Staubli VAL3: ros_server.pjx

--- ros_server.pjx ---
Parameters version=s7.7.2 stackSize=5000 millimeterUnit=true
Program file=dataReceiver.pgx
Program file=dataStreamer.pgx
Program file=decodeMsgBody.pgx
Program file=decodeMsgHeader.pgx
Program file=decTrajPt.pgx
Program file=decTrajPtFull.pgx
Program file=encodeAck.pgx
Program file=encodeJState.pgx
Program file=encodeStatus.pgx
Program file=encPrefixHeader.pgx
Program file=encTrajPtAck.pgx
Program file=encTrajPtFAck.pgx
Program file=fetchStatus.pgx
Program file=initParams.pgx
Program file=motionControl.pgx
Program file=pushMotion.pgx
Program file=recvData.pgx
Program file=recvHeartbeat.pgx
Program file=recvMsgBody.pgx
Program file=recvMsgHeader.pgx
Program file=recvTrajPt.pgx
Program file=recvTrajPtFull.pgx
Program file=screenUpdate.pgx
Program file=sendAck.pgx
Program file=sendData.pgx
Program file=sendRosMsg.pgx
Program file=setupRosMsgs.pgx
Program file=start.pgx
Program file=stop.pgx
Program file=toJointArrayRad.pgx
Program file=toJointRxDeg.pgx
Data file=ros_server.dtx
Library alias=libQueueFuncs path=Disk://ros_libs/QueueFuncs/QueueFuncs.pjx
Type name=RosSimpleMsg path=Disk://ros_libs/RosSimpleMsg/RosSimpleMsg.pjx
Type name=RobotStatusMsg path=Disk://ros_libs/RobotStatusMsg/RobotStatusMsg.pjx
Type name=JointStateMsg path=Disk://ros_libs/JointStateMsg/JointStateMsg.pjx
Type name=JointTrajPtMsg path=Disk://ros_libs/JointTrajPtMsg/JointTrajPtMsg.pjx
Type name=JointTrajPtFMsg path=Disk://ros_libs/JointTrajPtFMsg/JointTrajPtFMsg.pjx
Type name=JointFbkMsg path=Disk://ros_libs/JointFbkMsg/JointFbkMsg.pjx
Type name=MotionCmd path=Disk://ros_libs/MotionCmd/MotionCmd.pjx
Type name=Header path=Disk://ros_libs/Header/Header.pjx
Type name=Prefix path=Disk://ros_libs/Prefix/Prefix.pjx
Type name=Body path=Disk://ros_libs/Body/Body.pjx
Type name=Queue path=Disk://ros_libs/Queue/Queue.pjx

--- ros_server.dtx ---
public bool bFbkOverrun
public bool bMotionOverrun
public jointRx jCurrPose
public num nCounter
public num nFbkPeriod = 0.032
num nMotionPeriod = 0.012
public sio siTcpIpFbk = {link=Socket\Feedback}
public sio siTcpIpMotion = {link=Socket\Motion}
public string sStreamTaskName = "publisher"
public string sMotionTaskName
public bool bSendData
public RosSimpleMsg rosGenericMsg
  [0]
    Header header
      [0]
        num nMsgType
        num nCommType
        num nReplyCode
        num nData[12]
    Prefix prefix
      [0]
        num nLength
        num nData[4]
public jointRx jDesiredPose
public tool tTool = {fatherId=flange[0], ioLink=valve1}
public string sTrajPtTaskName
public bool bTrajPtOverrun
public RobotStatusMsg rosStatusMsg
  [0]
    Body body
      [0]
        num nData[28]
    Header header
      [0]
        num nMsgType
        num nCommType
        num nReplyCode
        num nData[12]
    Prefix prefix
      [0]
        num nLength
        num nData[4]
    RobotStatus robotStatus
      [0]
        num nDrivesPowered
        num nEStopped
        num nErrorCode
        num nInError
        num nInMotion
        num nMode
        num nMotionPossible
public JointStateMsg rosJointMsg
  [0]
    Header header
      [0]
        num nMsgType
        num nCommType
        num nReplyCode
        num nData[12]
    Body body
      [0]
        num nData[44]
    JointState jointState
      [0]
        num nSeq
        num nJoints[10]
    Prefix prefix
      [0]
        num nLength
        num nData[4]
public JointTrajPtMsg rosTrajPtMsg
  [0]
    Header header
      [0]
        num nMsgType
        num nCommType
        num nReplyCode
        num nData[12]
    JointTrajPt jointTrajPt
      [0]
        num nSeq
        num nJoints[10]
        num nVelocity
        num nDuration
    Prefix prefix
      [0]
        num nLength
        num nData[4]
    Body body
      [0]
        num nData[52]
public bool bRecvData
public JointTrajPtFMsg rosTrajPtFMsg
  [0]
    Header header
      [0]
        num nMsgType
        num nCommType
        num nReplyCode
        num nData[12]
    Prefix prefix
      [0]
        num nLength
        num nData[4]
    JointTrajPtFull jointTrajPtFull
      [0]
        num nRobotId
        num nSeq
        num nValidFields
        num nTime
        num nPositions[10]
        num nVelocities[10]
        num nAccelerations[10]
    Body body
      [0]
        num nData[136]
public JointFbkMsg rosJointFbkMsg
  [0]
    Header header
      [0]
        num nMsgType
        num nCommType
        num nReplyCode
        num nData[12]
    Prefix prefix
      [0]
        num nLength
        num nData[4]
    JointFeedback jointFeedback
      [0]
        num nRobotId
        num nValidFields
        num nTime
        num nPositions[10]
        num nVelocities[10]
        num nAccelerations[10]
    Body body
      [0]
        num nData[132]
public JointTrajPtFMsg rosTrajPtFAck
  [0]
    Header header
      [0]
        num nMsgType
        num nCommType
        num nReplyCode
        num nData[12]
    Prefix prefix
      [0]
        num nLength
        num nData[4]
    JointTrajPtFull jointTrajPtFull
      [0]
        num nRobotId
        num nSeq
        num nValidFields
        num nTime
        num nPositions[10]
        num nVelocities[10]
        num nAccelerations[10]
    Body body
      [0]
        num nData[136]
public JointTrajPtMsg rosTrajPtAck
  [0]
    Header header
      [0]
        num nMsgType
        num nCommType
        num nReplyCode
        num nData[12]
    JointTrajPt jointTrajPt
      [0]
        num nSeq
        num nJoints[10]
        num nVelocity
        num nDuration
    Prefix prefix
      [0]
        num nLength
        num nData[4]
    Body body
      [0]
        num nData[52]
public bool bScreenOverrun
public string sScreenTaskName
public num nScreenUpdate
public num nTrajReception
public num nInConnFlag
public num nOutConnFlag
public num nDebugStatus
public screen scDebug
public screen scMonitor
public string sHtbtTaskName
public num nMsgRecvState
public num nPtsPopped
public bool bStopNow
public MotionBuffer mTrajPt
  [0]
    mdesc mDesc = {leave=0, reach=0}
    num nDuration
    num nSequence
    jointRx jJointRx
public num nMotionProgress
public num nMoveId
public num nMovePts
public num nElapsedTime
public num nHeaderTime
public num nOtherTime
public num nStartTime
public bool bOverwriteVel
public num nKey

--- start.pgx ---
program start()
  local num l_nFbkPeriod
  local num l_nMotionPeriod
  local num l_nTrajPeriod
  local num l_nScreenUpdate
begin
  // Copyright (c) 2016, Ocado Technology - Robotics Research Team
  //
  // Licensed under the Apache License, Version 2.0 (the "License");
  // you may not use this file except in compliance with the License.
  // You may obtain a copy of the License at
  //
  //     http://www.apache.org/licenses/LICENSE-2.0
  //
  // Unless required by applicable law or agreed to in writing, software
  // distributed under the License is distributed on an "AS IS" BASIS,
  // WITHOUT WARRANTIES OR CONDITIONS OF ANY KIND, either express or implied.
  // See the License for the specific language governing permissions and
  // limitations under the License.



  // feedback task will run every 20ms (50Hz)
  l_nFbkPeriod=0.02
  //l_nFbkPeriod = 0.032 // 30Hz
  //l_nFbkPeriod = 0.05  // 20Hz
  //l_nFbkPeriod = 1.0   //  1Hz

  // motion control task will run every 4ms (250Hz)
  l_nMotionPeriod = 0.004
  //l_nMotionPeriod=0.012  // 83Hz
  //l_nMotionPeriod = 0.05 // 20Hz

  // data (trajectory) reception task will run every 4ms (250Hz)
  l_nTrajPeriod = 0.004
  // not in use at the moment
  l_nScreenUpdate = 1.0

  sStreamTaskName = "streamerTask"
  sTrajPtTaskName = "trajPtTask"
  sMotionTaskName = "motionTask"
  sScreenTaskName = "screenTask"
  sHtbtTaskName = "htbtTask"

  // initialise TCP/IP parameters
  call initParams()
  // setup prefix and header of ROS messages
  call setupRosMsgs()

  // socket connection status flags: initially disconnected
  nInConnFlag = 0
  nOutConnFlag = 0

  // flag defining whether velocity to be overwritten to max. vel.
  bOverwriteVel = false

  nPtsPopped = 0
  nMovePts = 0

  // flush buffer of incoming socket
  clearBuffer(siTcpIpMotion)
  // flush buffer of outgoing socket
  clearBuffer(siTcpIpFbk)

  // check if robot is not in emergency stop and wait until estop is reset
  if (esStatus() == 2)
    popUpMsg("Please reset E-Stop")
    wait(esStatus() < 2)
  endIf

  // before anything else, enable power (only works if robot is in remote mode)
  if (!isPowered())
    if (workingMode() >= 4)
      do
        enablePower()
        delay(2)
      until isPowered()
    else
      popUpMsg("Power must be enabled manually")
    endIf
  endIf

  // reset motion, potentially setting a start joint position for calling autoConnect() in the future
  resetMotion()

  // create joint state and robot status streamer task to send data to industrial_robot_client
  taskCreateSync sStreamTaskName, l_nFbkPeriod, bFbkOverrun, dataStreamer()

  // create trajectory point task to receive data from industrial_robot_client
  taskCreateSync sTrajPtTaskName, l_nTrajPeriod, bTrajPtOverrun, dataReceiver()
  //taskCreate sTrajPtTaskName, 100, dataReceiver()

  // create motion task to synchronously apply motion commands to robot
  taskCreateSync sMotionTaskName, l_nMotionPeriod, bMotionOverrun, motionControl()

  // create synchronous task to update screen
  //taskCreateSync sScreenTaskName, l_nScreenUpdate, bScreenOverrun, screenUpdate()
  taskCreate sScreenTaskName, 10, screenUpdate()

  // create asynchronous task to receive heartbeat on port 11002
  taskCreate sHtbtTaskName, 10, recvHeartbeat()

end

--- dataReceiver.pgx ---
public program dataReceiver()
  local num l_nStartTime
  local num l_nMsgRecvState
begin
  // Copyright (c) 2016, Ocado Technology - Robotics Research Team
  //
  // Licensed under the Apache License, Version 2.0 (the "License");
  // you may not use this file except in compliance with the License.
  // You may obtain a copy of the License at
  //
  //     http://www.apache.org/licenses/LICENSE-2.0
  //
  // Unless required by applicable law or agreed to in writing, software
  // distributed under the License is distributed on an "AS IS" BASIS,
  // WITHOUT WARRANTIES OR CONDITIONS OF ANY KIND, either express or implied.
  // See the License for the specific language governing permissions and
  // limitations under the License.



  // state machine at initial state
  // 0: receive header
  // 1: decode header
  // 2: receive body
  // 3: decode body
  // 4: push motion into buffer
  // 5: send ACK
  l_nMsgRecvState=0

  while (true)
    // usually for state machines a switch-case statement is a neat implementation
    // HOWEVER, at every iteration of while() this task is sequenced and only called
    // after whatever ms is was defined when created.
    // As a result, receiving one single message, pushing motion and sending ACK
    // would take 6 * task period using switch-case statement.
    // The desirable behaviour is to receive and decode a full message, push motion
    // into buffer and then send ACK to client WITHIN ONE ITERATION of while(),
    // hence the if statement sequence below
    l_nStartTime = clock()
    if (l_nMsgRecvState==0)
      call recvMsgHeader(l_nMsgRecvState)
    endIf
    nHeaderTime = clock() - l_nStartTime
    if (l_nMsgRecvState==1)
      call decodeMsgHeader(l_nMsgRecvState)
    endIf
    if (l_nMsgRecvState==2)
      call recvMsgBody(l_nMsgRecvState)
    endIf
    if (l_nMsgRecvState==3)
      call decodeMsgBody(l_nMsgRecvState)
    endIf
    if (l_nMsgRecvState==4)
      call pushMotion(l_nMsgRecvState)
    endIf
    if (l_nMsgRecvState==5)
      call encodeAck()
      call sendAck(l_nMsgRecvState)
    endIf
    nElapsedTime = clock() - l_nStartTime - nHeaderTime

    // assert state machine is working OK
    if (l_nMsgRecvState<0 or l_nMsgRecvState>5)
      popUpMsg("Data reception state machine error")
    endIf

    // sequence task
    delay(0)


  endWhile
end

--- dataStreamer.pgx ---
public program dataStreamer()
  local num l_nThrottle
  local jointRx l_jCurrPose
begin
  // Copyright (c) 2016, Ocado Technology - Robotics Research Team
  //
  // Licensed under the Apache License, Version 2.0 (the "License");
  // you may not use this file except in compliance with the License.
  // You may obtain a copy of the License at
  //
  //     http://www.apache.org/licenses/LICENSE-2.0
  //
  // Unless required by applicable law or agreed to in writing, software
  // distributed under the License is distributed on an "AS IS" BASIS,
  // WITHOUT WARRANTIES OR CONDITIONS OF ANY KIND, either express or implied.
  // See the License for the specific language governing permissions and
  // limitations under the License.



  l_nThrottle = 0
  while (true)
    // only attempt to send data if flag indicates that connection is established
    if (nOutConnFlag == 1)
      // fetch current joint positions
      l_jCurrPose=herej()
      // encode and send ROS simple_message ID 10: joint state
      call encodeJState(l_jCurrPose)
      call sendRosMsg(siTcpIpFbk, rosJointMsg.prefix, rosJointMsg.header, rosJointMsg.body, nOutConnFlag)

      // send Robot Status messages 5 times slower than Joint State
      if (l_nThrottle == 5)
        // fetch robot status
        call fetchStatus()
        // encode and send ROS simple_message ID 13: robot status
        call encodeStatus()
        call sendRosMsg(siTcpIpFbk, rosStatusMsg.prefix, rosStatusMsg.header, rosStatusMsg.body, nOutConnFlag)
        l_nThrottle = 0
      endIf
      l_nThrottle = l_nThrottle + 1
    else
      delay(0.1)
    endIf

    // sequence task
    delay(0)
  endWhile
end

--- decodeMsgBody.pgx ---
public program decodeMsgBody(num& x_nMsgRecvState)
  local bool l_bFlag
begin
  // Copyright (c) 2016, Ocado Technology - Robotics Research Team
  //
  // Licensed under the Apache License, Version 2.0 (the "License");
  // you may not use this file except in compliance with the License.
  // You may obtain a copy of the License at
  //
  //     http://www.apache.org/licenses/LICENSE-2.0
  //
  // Unless required by applicable law or agreed to in writing, software
  // distributed under the License is distributed on an "AS IS" BASIS,
  // WITHOUT WARRANTIES OR CONDITIONS OF ANY KIND, either express or implied.
  // See the License for the specific language governing permissions and
  // limitations under the License.



  l_bFlag=false

  switch rosGenericMsg.header.nMsgType
    case 11
      call decTrajPt(l_bFlag)
    break
    case 14
      call decTrajPtFull(l_bFlag)
    break
    default
    break
  endSwitch

  if (l_bFlag == true)
    // move on to state 4: push motion into buffer
    x_nMsgRecvState=4
  else
    // error whilst decoding msg body...
    if (rosGenericMsg.header.nCommType==2)
      switch rosGenericMsg.header.nMsgType
        case 11
          rosTrajPtAck.header.nReplyCode=2
        break
        case 14
          rosTrajPtFAck.header.nReplyCode=2
        break
        default
        break
      endSwitch
      // jump to state 5: sendAck()
      x_nMsgRecvState=5
    else
      // reset state machine, since no ACK is required
      x_nMsgRecvState=0
    endIf
  endIf
end

--- decodeMsgHeader.pgx ---
public program decodeMsgHeader(num& x_nMsgRecvState)
  local num l_nRetVal
begin
  // Copyright (c) 2016, Ocado Technology - Robotics Research Team
  //
  // Licensed under the Apache License, Version 2.0 (the "License");
  // you may not use this file except in compliance with the License.
  // You may obtain a copy of the License at
  //
  //     http://www.apache.org/licenses/LICENSE-2.0
  //
  // Unless required by applicable law or agreed to in writing, software
  // distributed under the License is distributed on an "AS IS" BASIS,
  // WITHOUT WARRANTIES OR CONDITIONS OF ANY KIND, either express or implied.
  // See the License for the specific language governing permissions and
  // limitations under the License.



  // decode message into generic message first
  l_nRetVal=fromBinary(rosGenericMsg.prefix.nData,4,"-4l",rosGenericMsg.prefix.nLength)
  if (l_nRetVal!=1)
    // error decoding prefix, reset state machine
    x_nMsgRecvState=0
    return
  endIf
  l_nRetVal=fromBinary(rosGenericMsg.header.nData,4,"-4l",rosGenericMsg.header.nMsgType)
  if (l_nRetVal!=1)
    // error decoding header (msg type), reset state machine
    x_nMsgRecvState=0
    return
  endIf
  l_nRetVal=fromBinary(rosGenericMsg.header.nData[4],4,"-4l",rosGenericMsg.header.nCommType)
  if (l_nRetVal!=1)
    // error decoding header (comm type), reset state machine
    x_nMsgRecvState=0
    return
  endIf
  l_nRetVal=fromBinary(rosGenericMsg.header.nData[8],4,"-4l",rosGenericMsg.header.nReplyCode)
  if (l_nRetVal!=1)
    // error decoding header (reply code), reset state machine
    x_nMsgRecvState=0
    return
  endIf

  // no errors detected whilst decoding prefix and header
  // move on to state 2: receive msg body
  x_nMsgRecvState=2
end

--- decTrajPt.pgx ---
public program decTrajPt(bool& x_bFlag (dimensions=1))
  local num l_nIndex
  local num l_nRetVal
begin
  // Copyright (c) 2016, Ocado Technology - Robotics Research Team
  //
  // Licensed under the Apache License, Version 2.0 (the "License");
  // you may not use this file except in compliance with the License.
  // You may obtain a copy of the License at
  //
  //     http://www.apache.org/licenses/LICENSE-2.0
  //
  // Unless required by applicable law or agreed to in writing, software
  // distributed under the License is distributed on an "AS IS" BASIS,
  // WITHOUT WARRANTIES OR CONDITIONS OF ANY KIND, either express or implied.
  // See the License for the specific language governing permissions and
  // limitations under the License.



  // decode message ID 11 body (data)

  // assume failure to decode
  rosTrajPtAck.header.nReplyCode=2

  // sequence
  l_nRetVal=fromBinary(rosTrajPtMsg.body.nData,4,"-4l",rosTrajPtMsg.jointTrajPt.nSeq)
  if (l_nRetVal!=1)
    x_bFlag=false
    return
  endIf

  // joints[10]
  for l_nIndex=0 to 9 step 1
    l_nRetVal=fromBinary(rosTrajPtMsg.body.nData[(l_nIndex*4)+4],4,"4.0l",rosTrajPtMsg.jointTrajPt.nJoints[l_nIndex])
    if (l_nRetVal!=1)
      x_bFlag=false
      return
    endIf
  endFor

  // velocity
  l_nRetVal=fromBinary(rosTrajPtMsg.body.nData[44],4,"4.0l",rosTrajPtMsg.jointTrajPt.nVelocity)
  if (l_nRetVal!=1)
    x_bFlag=false
    return
  endIf

  // duration
  l_nRetVal=fromBinary(rosTrajPtMsg.body.nData[48],4,"4.0l",rosTrajPtMsg.jointTrajPt.nDuration)
  if (l_nRetVal!=1)
    x_bFlag=false
    return
  endIf

  // decoding successful
  rosTrajPtAck.header.nReplyCode=1
  rosTrajPtAck.jointTrajPt.nSeq=rosTrajPtMsg.jointTrajPt.nSeq
  x_bFlag=true
end

--- decTrajPtFull.pgx ---
public program decTrajPtFull(bool& x_bFlag (dimensions=1))
  local num l_nIndex
  local num l_nRetVal
begin
  // Copyright (c) 2016, Ocado Technology - Robotics Research Team
  //
  // Licensed under the Apache License, Version 2.0 (the "License");
  // you may not use this file except in compliance with the License.
  // You may obtain a copy of the License at
  //
  //     http://www.apache.org/licenses/LICENSE-2.0
  //
  // Unless required by applicable law or agreed to in writing, software
  // distributed under the License is distributed on an "AS IS" BASIS,
  // WITHOUT WARRANTIES OR CONDITIONS OF ANY KIND, either express or implied.
  // See the License for the specific language governing permissions and
  // limitations under the License.



  // decode message ID 14 body (data)

  // assume failure to decode
  rosTrajPtFAck.header.nReplyCode=2

  // robotId
  l_nRetVal=fromBinary(rosTrajPtFMsg.body.nData,4,"-4l",rosTrajPtFMsg.jointTrajPtFull.nRobotId)
  if (l_nRetVal!=1)
    x_bFlag=false
    return
  endIf

  // sequence
  l_nRetVal=fromBinary(rosTrajPtFMsg.body.nData,4,"-4l",rosTrajPtFMsg.jointTrajPtFull.nSeq)
  if (l_nRetVal!=1)
    x_bFlag=false
    return
  endIf

  // valid fields
  l_nRetVal=fromBinary(rosTrajPtFMsg.body.nData,4,"-4l",rosTrajPtFMsg.jointTrajPtFull.nValidFields)
  if (l_nRetVal!=1)
    x_bFlag=false
    return
  endIf

  // time
  l_nRetVal=fromBinary(rosTrajPtFMsg.body.nData,4,"4.0l",rosTrajPtFMsg.jointTrajPtFull.nTime)
  if (l_nRetVal!=1)
    x_bFlag=false
    return
  endIf

  // positions[10]
  for l_nIndex=0 to 9 step 1
    l_nRetVal=fromBinary(rosTrajPtFMsg.body.nData[(l_nIndex*4)+16],4,"4.0l",rosTrajPtFMsg.jointTrajPtFull.nPositions[l_nIndex])
    if (l_nRetVal!=1)
      x_bFlag=false
      return
    endIf
  endFor

  // velocities[10]
  for l_nIndex=0 to 9 step 1
    l_nRetVal=fromBinary(rosTrajPtFMsg.body.nData[(l_nIndex*4)+56],4,"4.0l",rosTrajPtFMsg.jointTrajPtFull.nVelocities[l_nIndex])
    if (l_nRetVal!=1)
      x_bFlag=false
      return
    endIf
  endFor

  // accelerations[10]
  for l_nIndex=0 to 9 step 1
    l_nRetVal=fromBinary(rosTrajPtFMsg.body.nData[(l_nIndex*4)+96],4,"4.0l",rosTrajPtFMsg.jointTrajPtFull.nAccelerations[l_nIndex])
    if (l_nRetVal!=1)
      x_bFlag=false
      return
    endIf
  endFor

  // decoding successful
  rosTrajPtFAck.header.nReplyCode=1
  rosTrajPtFAck.jointTrajPtFull.nSeq=rosTrajPtFMsg.jointTrajPtFull.nSeq
  x_bFlag=true
end

--- encodeAck.pgx ---
public program encodeAck()
begin
  // Copyright (c) 2016, Ocado Technology - Robotics Research Team
  //
  // Licensed under the Apache License, Version 2.0 (the "License");
  // you may not use this file except in compliance with the License.
  // You may obtain a copy of the License at
  //
  //     http://www.apache.org/licenses/LICENSE-2.0
  //
  // Unless required by applicable law or agreed to in writing, software
  // distributed under the License is distributed on an "AS IS" BASIS,
  // WITHOUT WARRANTIES OR CONDITIONS OF ANY KIND, either express or implied.
  // See the License for the specific language governing permissions and
  // limitations under the License.



  switch rosGenericMsg.header.nMsgType
    case 11
      call encTrajPtAck()
    break
    case 14
      call encTrajPtFAck()
    break
    default
    break
  endSwitch
end

--- encodeJointFbk.pgx ---
public program encodeJointFbk()
  local num l_nRetVal
begin

end

--- encodeJState.pgx ---
public program encodeJState(jointRx& x_jCurrPose)
begin
  // Copyright (c) 2016, Ocado Technology - Robotics Research Team
  //
  // Licensed under the Apache License, Version 2.0 (the "License");
  // you may not use this file except in compliance with the License.
  // You may obtain a copy of the License at
  //
  //     http://www.apache.org/licenses/LICENSE-2.0
  //
  // Unless required by applicable law or agreed to in writing, software
  // distributed under the License is distributed on an "AS IS" BASIS,
  // WITHOUT WARRANTIES OR CONDITIONS OF ANY KIND, either express or implied.
  // See the License for the specific language governing permissions and
  // limitations under the License.



  // encode 'prefix' and 'header'
  call encPrefixHeader(rosJointMsg.prefix, rosJointMsg.header)

  // encode 'sequence' variable of body message (data)
  toBinary(rosJointMsg.jointState.nSeq,1,"-4l",rosJointMsg.body.nData)

  call toJointArrayRad(x_jCurrPose, rosJointMsg.jointState.nJoints)

  // encode 10 values representing joints[10]
  toBinary(rosJointMsg.jointState.nJoints,10,"4.0l",rosJointMsg.body.nData[4])
end

--- encodeStatus.pgx ---
public program encodeStatus()
begin
  // Copyright (c) 2016, Ocado Technology - Robotics Research Team
  //
  // Licensed under the Apache License, Version 2.0 (the "License");
  // you may not use this file except in compliance with the License.
  // You may obtain a copy of the License at
  //
  //     http://www.apache.org/licenses/LICENSE-2.0
  //
  // Unless required by applicable law or agreed to in writing, software
  // distributed under the License is distributed on an "AS IS" BASIS,
  // WITHOUT WARRANTIES OR CONDITIONS OF ANY KIND, either express or implied.
  // See the License for the specific language governing permissions and
  // limitations under the License.



  // encode 'prefix' and 'header'
  call encPrefixHeader(rosStatusMsg.prefix, rosStatusMsg.header)

  // encode variables of body message (data)
  toBinary(rosStatusMsg.robotStatus.nDrivesPowered,1,"-4l",rosStatusMsg.body.nData)
  toBinary(rosStatusMsg.robotStatus.nEStopped,1,"-4l",rosStatusMsg.body.nData[4])
  toBinary(rosStatusMsg.robotStatus.nErrorCode,1,"-4l",rosStatusMsg.body.nData[8])
  toBinary(rosStatusMsg.robotStatus.nInError,1,"-4l",rosStatusMsg.body.nData[12])
  toBinary(rosStatusMsg.robotStatus.nInMotion,1,"-4l",rosStatusMsg.body.nData[16])
  toBinary(rosStatusMsg.robotStatus.nMode,1,"-4l",rosStatusMsg.body.nData[20])
  toBinary(rosStatusMsg.robotStatus.nMotionPossible,1,"-4l",rosStatusMsg.body.nData[24])
end

--- encPrefixHeader.pgx ---
public program encPrefixHeader(Prefix& x_pPrefix, Header& x_hHeader)
begin
  // Copyright (c) 2016, Ocado Technology - Robotics Research Team
  //
  // Licensed under the Apache License, Version 2.0 (the "License");
  // you may not use this file except in compliance with the License.
  // You may obtain a copy of the License at
  //
  //     http://www.apache.org/licenses/LICENSE-2.0
  //
  // Unless required by applicable law or agreed to in writing, software
  // distributed under the License is distributed on an "AS IS" BASIS,
  // WITHOUT WARRANTIES OR CONDITIONS OF ANY KIND, either express or implied.
  // See the License for the specific language governing permissions and
  // limitations under the License.



  // encode prefix length
  toBinary(x_pPrefix.nLength,1,"-4l",x_pPrefix.nData)

  // encode header data
  toBinary(x_hHeader.nMsgType,1,"-4l",x_hHeader.nData)
  toBinary(x_hHeader.nCommType,1,"-4l",x_hHeader.nData[4])
  toBinary(x_hHeader.nReplyCode,1,"-4l",x_hHeader.nData[8])
end

--- encTrajPtAck.pgx ---
public program encTrajPtAck()
begin
  // Copyright (c) 2016, Ocado Technology - Robotics Research Team
  //
  // Licensed under the Apache License, Version 2.0 (the "License");
  // you may not use this file except in compliance with the License.
  // You may obtain a copy of the License at
  //
  //     http://www.apache.org/licenses/LICENSE-2.0
  //
  // Unless required by applicable law or agreed to in writing, software
  // distributed under the License is distributed on an "AS IS" BASIS,
  // WITHOUT WARRANTIES OR CONDITIONS OF ANY KIND, either express or implied.
  // See the License for the specific language governing permissions and
  // limitations under the License.



  // encode 'prefix' and 'header'
  call encPrefixHeader(rosTrajPtAck.prefix, rosTrajPtAck.header)

  // encode 'sequence' variable of body message (data)
  toBinary(rosTrajPtAck.jointTrajPt.nSeq,1,"-4l",rosTrajPtAck.body.nData)

  // encodings of 'joints[10]', 'velocity' and 'duration' ignored to save CPU time, since values are all zeros
end

--- encTrajPtFAck.pgx ---
public program encTrajPtFAck()
begin
  // Copyright (c) 2016, Ocado Technology - Robotics Research Team
  //
  // Licensed under the Apache License, Version 2.0 (the "License");
  // you may not use this file except in compliance with the License.
  // You may obtain a copy of the License at
  //
  //     http://www.apache.org/licenses/LICENSE-2.0
  //
  // Unless required by applicable law or agreed to in writing, software
  // distributed under the License is distributed on an "AS IS" BASIS,
  // WITHOUT WARRANTIES OR CONDITIONS OF ANY KIND, either express or implied.
  // See the License for the specific language governing permissions and
  // limitations under the License.



  // encode 'prefix' and 'header'
  call encPrefixHeader(rosTrajPtFAck.prefix, rosTrajPtFAck.header)

  // encode body message (data)
  toBinary(rosTrajPtFAck.jointTrajPtFull.nRobotId,1,"-4l",rosTrajPtFAck.body.nData)
  toBinary(rosTrajPtFAck.jointTrajPtFull.nSeq,1,"-4l",rosTrajPtFAck.body.nData[4])

  // encodings of 'positions[10]', velocities[10]' and accelerations[10]' ignored to save CPU time, since values are all zeros
end

--- fbkStreamer.pgx ---
public program fbkStreamer()
begin

end

--- fetchStatus.pgx ---
public program fetchStatus()
begin
  // Copyright (c) 2016, Ocado Technology - Robotics Research Team
  //
  // Licensed under the Apache License, Version 2.0 (the "License");
  // you may not use this file except in compliance with the License.
  // You may obtain a copy of the License at
  //
  //     http://www.apache.org/licenses/LICENSE-2.0
  //
  // Unless required by applicable law or agreed to in writing, software
  // distributed under the License is distributed on an "AS IS" BASIS,
  // WITHOUT WARRANTIES OR CONDITIONS OF ANY KIND, either express or implied.
  // See the License for the specific language governing permissions and
  // limitations under the License.



  // fetch robot status data

  // drives_powered
  if (isPowered()==true)
    rosStatusMsg.robotStatus.nDrivesPowered=1
  else
    rosStatusMsg.robotStatus.nDrivesPowered=0
  endIf

  // e-stopped
  if (esStatus()==2)
    rosStatusMsg.robotStatus.nEStopped=1
  else
    rosStatusMsg.robotStatus.nEStopped=0
  endIf

  // error_code
  if (taskStatus(sMotionTaskName) > 1)
    rosStatusMsg.robotStatus.nErrorCode = taskStatus(sMotionTaskName)
  elseIf (taskStatus(sTrajPtTaskName) > 1)
    rosStatusMsg.robotStatus.nErrorCode = taskStatus(sTrajPtTaskName)
  elseIf (taskStatus(sStreamTaskName) > 1)
    rosStatusMsg.robotStatus.nErrorCode = taskStatus(sStreamTaskName)
  elseIf (taskStatus(sHtbtTaskName) > 1)
    rosStatusMsg.robotStatus.nErrorCode = taskStatus(sHtbtTaskName)
  elseIf (taskStatus(sScreenTaskName) > 1)
    rosStatusMsg.robotStatus.nErrorCode = taskStatus(sScreenTaskName)
  else
    rosStatusMsg.robotStatus.nErrorCode = 0
  endIf

  // in_error
  if (taskStatus(sTrajPtTaskName) == 1 and taskStatus(sMotionTaskName) == 1 and taskStatus(sStreamTaskName) == 1 and taskStatus(sScreenTaskName) == 1 and taskStatus(sHtbtTaskName) == 1)
    rosStatusMsg.robotStatus.nInError = 0
  else
    rosStatusMsg.robotStatus.nInError = 1
  endIf

  // in_motion
  if (isSettled()==true)
    rosStatusMsg.robotStatus.nInMotion=0
  else
    rosStatusMsg.robotStatus.nInMotion=1
  endIf

  // mode (controller/pendant mode)
  // according to industrial_msgs/RobotMode, possible values are:
  // -1: unknown or unavailable
  //  1: teach or manual mode
  //  2: automatic mode (which I interpret as either local or remote)
  if (workingMode() == 0)
    rosStatusMsg.robotStatus.nMode = -1
  elseIf (workingMode()==1 or workingMode()==2)
    rosStatusMsg.robotStatus.nMode = 1
  elseIf (workingMode()==3 or workingMode()==4)
    rosStatusMsg.robotStatus.nMode = 2
  endIf

  // motion_possible:
  // drives must be powered and e-stop must be off
  // and dataReceiver and motionControl tasks must be
  // running normally
  if (isPowered() == true and esStatus() == 0 and taskStatus(sTrajPtTaskName) == 1 and taskStatus(sMotionTaskName) == 1)
    rosStatusMsg.robotStatus.nMotionPossible=1
  else
    rosStatusMsg.robotStatus.nMotionPossible=0
  endIf
end

--- initParams.pgx ---
public program initParams()
  local num l_nRetVal
begin
  // Copyright (c) 2016, Ocado Technology - Robotics Research Team
  //
  // Licensed under the Apache License, Version 2.0 (the "License");
  // you may not use this file except in compliance with the License.
  // You may obtain a copy of the License at
  //
  //     http://www.apache.org/licenses/LICENSE-2.0
  //
  // Unless required by applicable law or agreed to in writing, software
  // distributed under the License is distributed on an "AS IS" BASIS,
  // WITHOUT WARRANTIES OR CONDITIONS OF ANY KIND, either express or implied.
  // See the License for the specific language governing permissions and
  // limitations under the License.



  l_nRetVal=sioCtrl(siTcpIpMotion,"timeout",-1)
  if (l_nRetVal!=0)
    popUpMsg("Error while setting consumer timeout")
  endIf

  l_nRetVal=sioCtrl(siTcpIpFbk,"timeout",-1)
  if (l_nRetVal!=0)
    popUpMsg("Error while setting producer timeout")
  endIf
end

--- motionControl.pgx ---
public program motionControl()
  local MotionCmd l_mTrajPt
  local bool l_bFlag
  local MotionCmd l_motion
  local num l_nTime
  local bool l_bStopAndClean
  local num l_nElems
begin
  // Copyright (c) 2016, Ocado Technology - Robotics Research Team
  //
  // Licensed under the Apache License, Version 2.0 (the "License");
  // you may not use this file except in compliance with the License.
  // You may obtain a copy of the License at
  //
  //     http://www.apache.org/licenses/LICENSE-2.0
  //
  // Unless required by applicable law or agreed to in writing, software
  // distributed under the License is distributed on an "AS IS" BASIS,
  // WITHOUT WARRANTIES OR CONDITIONS OF ANY KIND, either express or implied.
  // See the License for the specific language governing permissions and
  // limitations under the License.



  nMoveId = -1

  while (true)
    // check connection status, and whether to stop motion
    if (nInConnFlag == 1 and nOutConnFlag == 1 and bStopNow == false)

      // process trajectory point from trajectory buffer
      call libQueueFuncs:getNumElems(qTrajPtBuffer, l_nElems)
      if (l_nElems > 0)
        call libQueueFuncs:pop(qTrajPtBuffer,l_mTrajPt, l_bFlag)
        if (l_bFlag == true)
          nPtsPopped = nPtsPopped + 1
          call libQueueFuncs:push(qMoveBuffer,l_mTrajPt,l_bFlag)
        endIf
      endIf

      // process motion command from move buffer
      // @TODO move buffer should have elements previously interpolated to ensure they are 4 ms apart
      call libQueueFuncs:getNumElems(qMoveBuffer, l_nElems)
      if (l_nElems > 0)
        call libQueueFuncs:pop(qMoveBuffer,l_motion,l_bFlag)
        if (l_bFlag == true)
          nMovePts = nMovePts + 1
          // contrary to what we did earlier, we unconditionally add the traj pt to the motion queue:
          // there doesn't appear to be a way to compare the 'current pose' of the robot to the pts
          // in the trajectory at the appropriate time (ie: when the robot is in motion and about to
          // start executing the segment towards 'l_motion').
          // Checking for dist(l_motion, herej()) (pseudo code) would not be correct as there will
          // always be a delay in the data coming out of herej() and the actual pose of the robot.
          // @TODO potentially set move id according to sequence value
          nMoveId = movej(l_motion.jJointRx, tTool, l_motion.mDesc)
        endIf
      endIf
    else
      // stop immediately -- resetMotion() also resets moveId
      resetMotion()
      // clear buffers
      call libQueueFuncs:clear(qTrajPtBuffer)
      call libQueueFuncs:clear(qMoveBuffer)
      bStopNow = false

      // debug
      nPtsPopped = 0
      nMovePts = 0
    endIf

    nMotionProgress = getMoveId()

    // sequence task
    delay(0)
  endWhile
end

--- pushMotion.pgx ---
public program pushMotion(num& x_nMsgRecvState)
  local bool l_bOk
  local num l_nCounter
  local num l_nJointError
  local MotionCmd l_mTrajPt
begin
  // Copyright (c) 2016, Ocado Technology - Robotics Research Team
  //
  // Licensed under the Apache License, Version 2.0 (the "License");
  // you may not use this file except in compliance with the License.
  // You may obtain a copy of the License at
  //
  //     http://www.apache.org/licenses/LICENSE-2.0
  //
  // Unless required by applicable law or agreed to in writing, software
  // distributed under the License is distributed on an "AS IS" BASIS,
  // WITHOUT WARRANTIES OR CONDITIONS OF ANY KIND, either express or implied.
  // See the License for the specific language governing permissions and
  // limitations under the License.



  switch rosGenericMsg.header.nMsgType
    case 11
      l_mTrajPt.nSequence=rosTrajPtMsg.jointTrajPt.nSeq

      // ROS joint position values are in rad, but VAL3 uses degrees
      call toJointRxDeg(rosTrajPtMsg.jointTrajPt.nJoints, l_mTrajPt.jJointRx)

      // from industrial_robot_client/src/joint_trajectory_interface.cpp
      // JointTrajectoryInterface::trajectory_to_msgs()
      // JointTrajectoryInterface::calc_speed()
      // velocity is converted to a scalar value representing % of max velocity,
      // such that 0.2 = 20% of maximum joint speed
      l_mTrajPt.mDesc.vel= limit((rosTrajPtMsg.jointTrajPt.nVelocity * 100), 0, 100)
      l_mTrajPt.nDuration=rosTrajPtMsg.jointTrajPt.nDuration

    break
    case 14
      l_mTrajPt.nSequence=rosTrajPtFMsg.jointTrajPtFull.nSeq
      l_mTrajPt.nDuration=rosTrajPtFMsg.jointTrajPtFull.nTime

      // ROS joint position values are in rad, but VAL3 uses degrees
      call toJointRxDeg(rosTrajPtFMsg.jointTrajPtFull.nPositions, l_mTrajPt.jJointRx)

      // from industrial_robot_client/src/joint_trajectory_interface.cpp
      // JointTrajectoryInterface::trajectory_to_msgs()
      // JointTrajectoryInterface::calc_speed()
      // velocity is converted to a scalar value representing % of max velocity,
      // such that 0.2 = 20% of maximum joint speed
      l_mTrajPt.mDesc.vel= limit((rosTrajPtFMsg.jointTrajPtFull.nVelocities[0] * 100), 0, 100)
      // not sure about accelerations as yet
      l_mTrajPt.mDesc.accel=rosTrajPtFMsg.jointTrajPtFull.nAccelerations[0]
      l_mTrajPt.mDesc.decel=l_mTrajPt.mDesc.accel
    break
    default
    break
  endSwitch

  // see github.com/ros-industrial/industrial_core/simple_message/include/simple_message/joint_traj_pt.h
  if (l_mTrajPt.nSequence==-4)
    // set flag to stop immediately
    bStopNow=true
  else
    // check whether velocity value should be overwritten with value set on teach pendant
    if (bOverwriteVel == true)
      // overwrite velocity (and acceleration - ?)
      l_mTrajPt.mDesc.vel = getMonitorSpeed()
      // explicitly setting accel and decel to VAL3 default values
      l_mTrajPt.mDesc.accel = 9999
      l_mTrajPt.mDesc.decel = 9999
    endIf
    // only push motion into buffer if not a STOP message
    // and if joint positions are within software joint limits
    // and if velocity is greater than zero (beucase movej() will not accept vel <= 0)
    if (isInRange(l_mTrajPt.jJointRx) and l_mTrajPt.mDesc.vel > 0)
      call libQueueFuncs:push(qTrajPtBuffer,l_mTrajPt,l_bOk)
    else
      l_bOk = false
    endIf

    if (l_bOk==false)
      // could not push trajectory point into buffer
      // thus ACK should flag FAILURE, but only if comm type is request
      if (rosGenericMsg.header.nCommType==2)
        switch rosGenericMsg.header.nMsgType
          case 11
            rosTrajPtAck.header.nReplyCode=2
          break
          case 14
            rosTrajPtFAck.header.nReplyCode=2
          break
          default
          break
        endSwitch
      endIf
    endIf
  endIf
  // check whether ACK should be sent
  if (rosGenericMsg.header.nCommType == 2)
    // comm type request requires ACK
    x_nMsgRecvState = 5
  else
    // other comm types (e.g., topic) does not require ACK, hence skip state
    x_nMsgRecvState = 0
  endIf
end

--- recvData.pgx ---
public program recvData(sio& x_sTcpSocket, num& x_nData[], num& x_nConnFlag, bool& x_bValidFlag)
  local num l_nByte
  local num l_nBytesRecv
  local num l_nIndex
begin
  // Copyright (c) 2016, Ocado Technology - Robotics Research Team
  //
  // Licensed under the Apache License, Version 2.0 (the "License");
  // you may not use this file except in compliance with the License.
  // You may obtain a copy of the License at
  //
  //     http://www.apache.org/licenses/LICENSE-2.0
  //
  // Unless required by applicable law or agreed to in writing, software
  // distributed under the License is distributed on an "AS IS" BASIS,
  // WITHOUT WARRANTIES OR CONDITIONS OF ANY KIND, either express or implied.
  // See the License for the specific language governing permissions and
  // limitations under the License.



  // attempt to receive data on specified socket

  // x_nConnFlag holds the current connection status of x_sTcpSocket

  l_nBytesRecv=0
  l_nIndex=0
  x_bValidFlag=false

  while (l_nBytesRecv<size(x_nData))
    l_nIndex=sioGet(x_sTcpSocket,l_nByte)
    if (l_nIndex==1)
      x_nData[l_nBytesRecv]=l_nByte
      l_nBytesRecv=l_nBytesRecv+1
      // received a byte, set flag to indicate connection
      x_nConnFlag=1
    elseIf (l_nIndex==-1)
      // error or timeout, indicate only if connection previously established
      if (x_nConnFlag==1)
        x_nConnFlag=-1
        // close connection properly (to avoid CLOSE_WAIT)
        clearBuffer(x_sTcpSocket)
      endIf
      return
    elseIf (l_nIndex == 0)
      // sioGet() returns 0 when connection is alive, thus set flag
      x_nConnFlag = 1
      if (l_nBytesRecv == 0)
        return
      endIf
    else
      // either < -1 or > 1
      popUpMsg("sioGet() returned " + toString("", l_nIndex))
      return
    endIf
  endWhile
  x_bValidFlag=true
end

--- recvHeartbeat.pgx ---
public program recvHeartbeat()
  local num l_nByte
  local num l_nBytesRecv
  local num l_nHtbt
  local num l_nHtbtB[4]
  local num l_nIndex
begin
  // Copyright (c) 2016, Ocado Technology - Robotics Research Team
  //
  // Licensed under the Apache License, Version 2.0 (the "License");
  // you may not use this file except in compliance with the License.
  // You may obtain a copy of the License at
  //
  //     http://www.apache.org/licenses/LICENSE-2.0
  //
  // Unless required by applicable law or agreed to in writing, software
  // distributed under the License is distributed on an "AS IS" BASIS,
  // WITHOUT WARRANTIES OR CONDITIONS OF ANY KIND, either express or implied.
  // See the License for the specific language governing permissions and
  // limitations under the License.



  while (true)
    l_nBytesRecv=0
    l_nIndex = sioGet(siTcpIpFbk, l_nByte)
    if (l_nIndex == -1)
      // connection not established or connection lost
      if (nOutConnFlag == 1)
        nOutConnFlag = -1
      endIf
    else
      // it means l_nIndex >= 0: connection established
      // check if connection had not already been established
      if (nOutConnFlag != 1)
        // delay data output to avoid sync issues with client
        delay(1.0)
        // flag connection as established
        nOutConnFlag = 1
      endIf
    endIf
  endWhile
end

--- recvMsgBody.pgx ---
public program recvMsgBody(num& x_nMsgRecvState)
  local bool l_bFlag
begin
  // Copyright (c) 2016, Ocado Technology - Robotics Research Team
  //
  // Licensed under the Apache License, Version 2.0 (the "License");
  // you may not use this file except in compliance with the License.
  // You may obtain a copy of the License at
  //
  //     http://www.apache.org/licenses/LICENSE-2.0
  //
  // Unless required by applicable law or agreed to in writing, software
  // distributed under the License is distributed on an "AS IS" BASIS,
  // WITHOUT WARRANTIES OR CONDITIONS OF ANY KIND, either express or implied.
  // See the License for the specific language governing permissions and
  // limitations under the License.



  l_bFlag=false

  switch rosGenericMsg.header.nMsgType
    case 11
      call recvTrajPt(l_bFlag)
    break
    case 14
      call recvTrajPtFull(l_bFlag)
    break
    default
    break
  endSwitch

  if (l_bFlag == true)
    // move on to state 3: decode msg body
    x_nMsgRecvState=3
  else
    // error whilst receiving msg body, reset state machine
    x_nMsgRecvState=0
  endIf
end

--- recvMsgHeader.pgx ---
public program recvMsgHeader(num& x_nMsgRecvState)
  local bool l_bFlag
begin
  // Copyright (c) 2016, Ocado Technology - Robotics Research Team
  //
  // Licensed under the Apache License, Version 2.0 (the "License");
  // you may not use this file except in compliance with the License.
  // You may obtain a copy of the License at
  //
  //     http://www.apache.org/licenses/LICENSE-2.0
  //
  // Unless required by applicable law or agreed to in writing, software
  // distributed under the License is distributed on an "AS IS" BASIS,
  // WITHOUT WARRANTIES OR CONDITIONS OF ANY KIND, either express or implied.
  // See the License for the specific language governing permissions and
  // limitations under the License.



  // attempt to receive message prefix and header
  call recvData(siTcpIpMotion,rosGenericMsg.prefix.nData,nInConnFlag,l_bFlag)
  if (l_bFlag == true)
    call recvData(siTcpIpMotion,rosGenericMsg.header.nData,nInConnFlag,l_bFlag)
  endIf

  if (l_bFlag == true)
    // move on to state 1: decode header
    x_nMsgRecvState=1
  else
    // error: reset state to 0: receive header
    x_nMsgRecvState=0
  endIf
end

--- recvTrajPt.pgx ---
public program recvTrajPt(bool& x_bFlag)
begin
  // Copyright (c) 2016, Ocado Technology - Robotics Research Team
  //
  // Licensed under the Apache License, Version 2.0 (the "License");
  // you may not use this file except in compliance with the License.
  // You may obtain a copy of the License at
  //
  //     http://www.apache.org/licenses/LICENSE-2.0
  //
  // Unless required by applicable law or agreed to in writing, software
  // distributed under the License is distributed on an "AS IS" BASIS,
  // WITHOUT WARRANTIES OR CONDITIONS OF ANY KIND, either express or implied.
  // See the License for the specific language governing permissions and
  // limitations under the License.



  // attempt to receive message ID 11 data (prefix and header are in rosGenericMsg)
  rosTrajPtMsg.prefix.nLength=rosGenericMsg.prefix.nLength
  rosTrajPtMsg.header.nMsgType=rosGenericMsg.header.nMsgType
  rosTrajPtMsg.header.nCommType=rosGenericMsg.header.nCommType
  rosTrajPtMsg.header.nReplyCode=rosGenericMsg.header.nReplyCode

  call recvData(siTcpIpMotion,rosTrajPtMsg.body.nData,nInConnFlag,x_bFlag)
end

--- recvTrajPtFull.pgx ---
public program recvTrajPtFull(bool& x_bFlag)
begin
  // Copyright (c) 2016, Ocado Technology - Robotics Research Team
  //
  // Licensed under the Apache License, Version 2.0 (the "License");
  // you may not use this file except in compliance with the License.
  // You may obtain a copy of the License at
  //
  //     http://www.apache.org/licenses/LICENSE-2.0
  //
  // Unless required by applicable law or agreed to in writing, software
  // distributed under the License is distributed on an "AS IS" BASIS,
  // WITHOUT WARRANTIES OR CONDITIONS OF ANY KIND, either express or implied.
  // See the License for the specific language governing permissions and
  // limitations under the License.



  // receive message ID 14 data (prefix and header are in rosGenericMsg)
  rosTrajPtFMsg.prefix.nLength=rosGenericMsg.prefix.nLength
  rosTrajPtFMsg.header.nMsgType=rosGenericMsg.header.nMsgType
  rosTrajPtFMsg.header.nCommType=rosGenericMsg.header.nCommType
  rosTrajPtFMsg.header.nReplyCode=rosGenericMsg.header.nReplyCode

  call recvData(siTcpIpMotion,rosTrajPtFMsg.body.nData,nInConnFlag,x_bFlag)
end

--- screenUpdate.pgx ---
public program screenUpdate()
  local num l_nKey
  local num l_nExecStatus
  local num l_nElems
begin
  // Copyright (c) 2016, Ocado Technology - Robotics Research Team
  //
  // Licensed under the Apache License, Version 2.0 (the "License");
  // you may not use this file except in compliance with the License.
  // You may obtain a copy of the License at
  //
  //     http://www.apache.org/licenses/LICENSE-2.0
  //
  // Unless required by applicable law or agreed to in writing, software
  // distributed under the License is distributed on an "AS IS" BASIS,
  // WITHOUT WARRANTIES OR CONDITIONS OF ANY KIND, either express or implied.
  // See the License for the specific language governing permissions and
  // limitations under the License.



  l_nExecStatus = 0
  userPage(scMonitor)
  cls(scMonitor)
  title(scMonitor, "ROS-I server")

  while (true)
    // clear screen
    cls(scMonitor)

    // toggle velocity overwrite upon release of F1 key
    l_nKey = getKey(scMonitor)
    call libQueueFuncs:getNumElems(qMoveBuffer,l_nElems)
    if (l_nKey == 277 and bOverwriteVel == false)
      if (l_nElems == 0)
        bOverwriteVel = true
      else
        popUpMsg("Motion buffer not empty; cannot enable V/OW")
      endIf
    elseIf (l_nKey == 278 and bOverwriteVel == true)
      if (l_nElems == 0)
        bOverwriteVel = false
      else
        popUpMsg("Motion buffer not empty; cannot disable V/OW")
      endIf
    endIf

    // update connection status on port 11000
    gotoxy(scMonitor, 0,0)
    // 11 characteres: gotoxy(12,0) to insert status
    put(scMonitor, "Port 11000:")
    gotoxy(scMonitor, 12,0)
    switch nInConnFlag
      case -1
        put(scMonitor, "connection lost")
      break
      case 0
        put(scMonitor, "not connected")
      break
      case 1
        put(scMonitor, "connected")
      break
      default
        put(scMonitor, "not connected")
      break
    endSwitch

    // update connection status on port 11002
    gotoxy(scMonitor, 0,1)
    // 11 characteres: gotoxy(12,1) to insert status
    put(scMonitor, "Port 11002:")
    gotoxy(scMonitor, 12,1)
    switch nOutConnFlag
      case -1
        put(scMonitor, "connection lost")
      break
      case 0
        put(scMonitor, "not connected")
      break
      case 1
        put(scMonitor, "connected")
      break
      default
        put(scMonitor, "not connected")
      break
    endSwitch

    // update trajectory buffer size
    call libQueueFuncs:getNumElems(qTrajPtBuffer,l_nElems)
    gotoxy(scMonitor, 0,3)
    // 18 characteres: gotoxy(19,3) to insert status
    put(scMonitor, "Trajectory buffer:")
    gotoxy(scMonitor, 19,3)
    put(scMonitor, l_nElems)
    // also print number of points popped from buffer
    gotoxy(scMonitor, 24,3)
    put(scMonitor, nPtsPopped)
    // do the same for move buffer
    call libQueueFuncs:getNumElems(qMoveBuffer,l_nElems)
    gotoxy(scMonitor, 0,4)
    put(scMonitor, "Motion buffer:")
    gotoxy(scMonitor, 19,4)
    put(scMonitor, l_nElems)
    gotoxy(scMonitor, 24,4)
    put(scMonitor, nMovePts)

    // display velocity overwrite status
    gotoxy(scMonitor, 0,5)
    put(scMonitor, "Velocity overwrite:")
    gotoxy(scMonitor, 20,5)
    if (bOverwriteVel == true)
      put(scMonitor, "enabled")
    else
      put(scMonitor, "disabled")
    endIf

    // display nMoveId and nMotionProgress
    gotoxy(scMonitor, 0,7)
    put(scMonitor, "moveId:")
    gotoxy(scMonitor, 8,7)
    put(scMonitor, nMoveId)
    gotoxy(scMonitor, 13,7)
    put(scMonitor, "progress:")
    gotoxy(scMonitor, 23,7)
    put(scMonitor, nMotionProgress)

    // display time between valid trajectory point received and ACK sent
    gotoxy(scMonitor, 0,9)
    put(scMonitor, "recvMsgHeader:")
    gotoxy(scMonitor, 15,9)
    put(scMonitor, toString(".4", nHeaderTime))

    gotoxy(scMonitor, 0,10)
    put(scMonitor, "other states:")
    gotoxy(scMonitor, 15,10)
    put(scMonitor, toString(".4", nElapsedTime))

    // update debug status
    gotoxy(scMonitor, 18,12)
    switch l_nExecStatus
      case 0
        put(scMonitor, "[+]")
        l_nExecStatus = 1
      break
      case 1
        put(scMonitor, "[-]")
        l_nExecStatus = 0
      break
      default
      break
    endSwitch

    // add Function keys labels
    gotoxy(scMonitor, 30,13)
    put(scMonitor, "V/ON")
    gotoxy(scMonitor, 35,13)
    put(scMonitor, "V/OFF")

    // sequence task
    //delay(0)
    delay(0.5)
  endWhile
end

--- sendAck.pgx ---
public program sendAck(num& x_nMsgRecvState)
begin
  // Copyright (c) 2016, Ocado Technology - Robotics Research Team
  //
  // Licensed under the Apache License, Version 2.0 (the "License");
  // you may not use this file except in compliance with the License.
  // You may obtain a copy of the License at
  //
  //     http://www.apache.org/licenses/LICENSE-2.0
  //
  // Unless required by applicable law or agreed to in writing, software
  // distributed under the License is distributed on an "AS IS" BASIS,
  // WITHOUT WARRANTIES OR CONDITIONS OF ANY KIND, either express or implied.
  // See the License for the specific language governing permissions and
  // limitations under the License.



  switch rosGenericMsg.header.nMsgType
    case 11
      call sendRosMsg(siTcpIpMotion, rosTrajPtAck.prefix, rosTrajPtAck.header, rosTrajPtAck.body, nInConnFlag)
    break
    case 14
      call sendRosMsg(siTcpIpMotion, rosTrajPtFAck.prefix, rosTrajPtFAck.header, rosTrajPtFAck.body, nInConnFlag)
    break
    default
    break
  endSwitch

  // regardless of result from sending ACK
  // reset state machine to receive new messages
  x_nMsgRecvState=0
end

--- sendData.pgx ---
public program sendData(sio& x_sTcpSocket, num& x_nData[], num& x_nFlag)
  local num l_nRetVal
begin
  // Copyright (c) 2016, Ocado Technology - Robotics Research Team
  //
  // Licensed under the Apache License, Version 2.0 (the "License");
  // you may not use this file except in compliance with the License.
  // You may obtain a copy of the License at
  //
  //     http://www.apache.org/licenses/LICENSE-2.0
  //
  // Unless required by applicable law or agreed to in writing, software
  // distributed under the License is distributed on an "AS IS" BASIS,
  // WITHOUT WARRANTIES OR CONDITIONS OF ANY KIND, either express or implied.
  // See the License for the specific language governing permissions and
  // limitations under the License.



  // send data via socket connection...
  // but only if connection is alive
  if (x_nFlag == 1)
    l_nRetVal=sioSet(x_sTcpSocket,x_nData)
    if (l_nRetVal==-1)
      if (x_nFlag==1)
        x_nFlag=-1
      endIf
    elseIf (l_nRetVal<size(x_nData))
      popUpMsg("Error while sending data")
      x_nFlag=-1
    endIf
  endIf
end

--- sendJointFbk.pgx ---
public program sendJointFbk()
  local num l_nRetVal
begin

end

--- sendJState.pgx ---
public program sendJState()
  local num l_nRetVal
begin
  call sendData(siTcpIpFbk,rosJointMsg.prefix.nData,nOutConnFlag)
  call sendData(siTcpIpFbk,rosJointMsg.header.nData,nOutConnFlag)
  call sendData(siTcpIpFbk,rosJointMsg.body.nData,nOutConnFlag)
end

--- sendRosMsg.pgx ---
public program sendRosMsg(sio& x_sTcpSocket, Prefix& x_pPrefix, Header& x_hHeader, Body& x_bBody, num& x_nConnFlag)
begin
  // Copyright (c) 2016, Ocado Technology - Robotics Research Team
  //
  // Licensed under the Apache License, Version 2.0 (the "License");
  // you may not use this file except in compliance with the License.
  // You may obtain a copy of the License at
  //
  //     http://www.apache.org/licenses/LICENSE-2.0
  //
  // Unless required by applicable law or agreed to in writing, software
  // distributed under the License is distributed on an "AS IS" BASIS,
  // WITHOUT WARRANTIES OR CONDITIONS OF ANY KIND, either express or implied.
  // See the License for the specific language governing permissions and
  // limitations under the License.



  call sendData(x_sTcpSocket, x_pPrefix.nData, x_nConnFlag)
  call sendData(x_sTcpSocket, x_hHeader.nData, x_nConnFlag)
  call sendData(x_sTcpSocket, x_bBody.nData, x_nConnFlag)
end

--- sendStatus.pgx ---
public program sendStatus()
  local num l_nRetVal
begin
  call sendData(siTcpIpFbk,rosStatusMsg.prefix.nData,nOutConnFlag)
  call sendData(siTcpIpFbk,rosStatusMsg.header.nData,nOutConnFlag)
  call sendData(siTcpIpFbk,rosStatusMsg.body.nData,nOutConnFlag)
end

--- sendTrajPtAck.pgx ---
public program sendTrajPtAck()
  local num l_nRetVal
begin
  // send message length (prefix)
  call sendData(siTcpIpMotion,rosTrajPtAck.prefix.nData,nInConnFlag)
  // send message header (msg type, comm type, reply code)
  call sendData(siTcpIpMotion,rosTrajPtAck.header.nData,nInConnFlag)
  call sendData(siTcpIpMotion,rosTrajPtAck.body.nData,nInConnFlag)
end

--- sendTrajPtFAck.pgx ---
public program sendTrajPtFAck()
  local num l_nRetVal
begin
  // send message length (prefix)
  call sendData(siTcpIpMotion,rosTrajPtFAck.prefix.nData,nInConnFlag)
  // send message header (msg type, comm type, reply code)
  call sendData(siTcpIpMotion,rosTrajPtFAck.header.nData,nInConnFlag)
  call sendData(siTcpIpMotion,rosTrajPtFAck.body.nData,nInConnFlag)
end

--- setupRosMsgs.pgx ---
public program setupRosMsgs()
begin
  // Copyright (c) 2016, Ocado Technology - Robotics Research Team
  //
  // Licensed under the Apache License, Version 2.0 (the "License");
  // you may not use this file except in compliance with the License.
  // You may obtain a copy of the License at
  //
  //     http://www.apache.org/licenses/LICENSE-2.0
  //
  // Unless required by applicable law or agreed to in writing, software
  // distributed under the License is distributed on an "AS IS" BASIS,
  // WITHOUT WARRANTIES OR CONDITIONS OF ANY KIND, either express or implied.
  // See the License for the specific language governing permissions and
  // limitations under the License.



  // Joint state message (ID 10)
  // prefix length = 12 + 44
  rosJointMsg.prefix.nLength=56
  rosJointMsg.header.nMsgType=10
  rosJointMsg.header.nCommType=1
  rosJointMsg.header.nReplyCode=0
  // sequence
  rosJointMsg.jointState.nSeq=0



  // Trajectory point message (ID 11)
  // prefix length = 12 + 52
  rosTrajPtAck.prefix.nLength=64
  rosTrajPtAck.header.nMsgType=11
  rosTrajPtAck.header.nCommType=3
  // reply: 1 = success, 2 = failure
  rosTrajPtAck.header.nReplyCode=1
  // joints are assumed to be initiliased to zero

  // the message bellow will be filled upon reception
  rosTrajPtMsg.prefix.nLength=64



  // Robot status message (ID 13)
  // prefix length = 12 + 28
  rosStatusMsg.prefix.nLength=40
  rosStatusMsg.header.nMsgType=13
  rosStatusMsg.header.nCommType=1
  rosStatusMsg.header.nReplyCode=0



  // Trajectory point full message (ID 14)
  // prefix length = 12 + 136
  rosTrajPtFAck.prefix.nLength=148
  rosTrajPtFAck.header.nMsgType=14
  rosTrajPtFAck.header.nCommType=3
  // reply: 1 = success, 2 = failure
  rosTrajPtFAck.header.nReplyCode=1
  // body (data) assumed to be initialised to zero

  // the message bellow will be filled upon reception
  rosTrajPtFMsg.prefix.nLength=148



  // Joint feedback message (ID 15)
  // prefix length = 12 + 132
  rosJointFbkMsg.prefix.nLength=144
  rosJointFbkMsg.header.nMsgType=15
  rosJointFbkMsg.header.nCommType=1
  rosJointFbkMsg.header.nReplyCode=0
end

--- stop.pgx ---
program stop()
begin
  // Copyright (c) 2016, Ocado Technology - Robotics Research Team
  //
  // Licensed under the Apache License, Version 2.0 (the "License");
  // you may not use this file except in compliance with the License.
  // You may obtain a copy of the License at
  //
  //     http://www.apache.org/licenses/LICENSE-2.0
  //
  // Unless required by applicable law or agreed to in writing, software
  // distributed under the License is distributed on an "AS IS" BASIS,
  // WITHOUT WARRANTIES OR CONDITIONS OF ANY KIND, either express or implied.
  // See the License for the specific language governing permissions and
  // limitations under the License.



  resetMotion()
  popUpMsg("Pending movement commands have been cancelled.")
  cls()
end

--- toJointArrayRad.pgx ---
public program toJointArrayRad(jointRx& x_jJointRx, num& x_nJointArray[])
  local num l_nDeg2Rad
begin
  // Copyright (c) 2016, Ocado Technology - Robotics Research Team
  //
  // Licensed under the Apache License, Version 2.0 (the "License");
  // you may not use this file except in compliance with the License.
  // You may obtain a copy of the License at
  //
  //     http://www.apache.org/licenses/LICENSE-2.0
  //
  // Unless required by applicable law or agreed to in writing, software
  // distributed under the License is distributed on an "AS IS" BASIS,
  // WITHOUT WARRANTIES OR CONDITIONS OF ANY KIND, either express or implied.
  // See the License for the specific language governing permissions and
  // limitations under the License.



  l_nDeg2Rad = 0.01745329251

  // assuming the remaining elements (6-9) have zeros assigned by default
  x_nJointArray[0] = x_jJointRx.j1 * l_nDeg2Rad
  x_nJointArray[1] = x_jJointRx.j2 * l_nDeg2Rad
  x_nJointArray[2] = x_jJointRx.j3 * l_nDeg2Rad
  x_nJointArray[3] = x_jJointRx.j4 * l_nDeg2Rad
  x_nJointArray[4] = x_jJointRx.j5 * l_nDeg2Rad
  x_nJointArray[5] = x_jJointRx.j6 * l_nDeg2Rad
end

--- toJointRxDeg.pgx ---
public program toJointRxDeg(num& x_nJointArray[], jointRx& x_jJointRx)
  local num l_nRad2Deg
begin
  // Copyright (c) 2016, Ocado Technology - Robotics Research Team
  //
  // Licensed under the Apache License, Version 2.0 (the "License");
  // you may not use this file except in compliance with the License.
  // You may obtain a copy of the License at
  //
  //     http://www.apache.org/licenses/LICENSE-2.0
  //
  // Unless required by applicable law or agreed to in writing, software
  // distributed under the License is distributed on an "AS IS" BASIS,
  // WITHOUT WARRANTIES OR CONDITIONS OF ANY KIND, either express or implied.
  // See the License for the specific language governing permissions and
  // limitations under the License.



  l_nRad2Deg = 57.2957795131

  x_jJointRx.j1 = x_nJointArray[0] * l_nRad2Deg
  x_jJointRx.j2 = x_nJointArray[1] * l_nRad2Deg
  x_jJointRx.j3 = x_nJointArray[2] * l_nRad2Deg
  x_jJointRx.j4 = x_nJointArray[3] * l_nRad2Deg
  x_jJointRx.j5 = x_nJointArray[4] * l_nRad2Deg
  x_jJointRx.j6 = x_nJointArray[5] * l_nRad2Deg
end
